(* CODESYS project xlh_transport_trolley_ST_00_90.project
   Description: Receives some incoming messages and echoes them with CAN-ID +1
   Company: 3S - Smart Software Solutions GmbH
   Version: 1.0.0.0
   Title: CAN Bus API Example
   Author: 3S - Smart Software Solutions GmbH

Project tree, tasks and I/O mapping:
  xlh_base : CODESYS Control for Raspberry Pi 64 SL, CODESYS, order no. 2302000009, version 4.18.0.0
    application app
      libraries: Standard, 3.5.18.0 (System); Util, 3.5.21.0 (System); VisuDialogs, * (System); Memory, * (3S - Smart Software Solutions GmbH); CmpBitmapPool, * (System)
      task MAIN_TASK (cyclic, interval 5 ms, priority 0) calls MAIN
      task VISU_TASK (cyclic, interval 100 ms, priority 31) calls VisuElems.Visu_Prg
      FSM/
        program TW_ST [ST]
        data type eTW
      visualisation VISU_SIMU
      function block FB_SIMU_TW [ST]
      image pool ImagePool
      program MAIN [ST]
      Depictor
      function block FB_XLH_GPIO [CFC]
    SoftMotion General Axis Pool
      a_axis : SM_Drive_PosControl, CODESYS, order no. 1805, version 4.18.0.0
          settings: wDriveID = 4; dwRatioTechUnitsDenom = 101846; iRatioTechUnitsNum = -125; eRampType = 1; fSWMaxVelocity = 50; fSWMaxAcceleration = 100; fSWMaxDeceleration = 100; fSWMaxJerk = 1000; fSWLimitNegative = -1000.0; ScalingIncs = 814768; ScalingUnits = 1000; InvertDirection = TRUE; IsLinearMotor = TRUE; MaximumOutputVelocityInt = 40738; MinimumOutputVelocityInt = -40738; Kp = 0.05; MaxFollowingError = 5.0; EnableFollowingErrorCheck = TRUE; DeadTime = 3.0
      x_axis : SM_Drive_PosControl, CODESYS, order no. 1805, version 4.18.0.0
          settings: dwRatioTechUnitsDenom = 101846; iRatioTechUnitsNum = 125; eRampType = 1; fSWMaxVelocity = 50; fSWMaxAcceleration = 100; fSWMaxDeceleration = 100; fSWMaxJerk = 1000; fSWLimitNegative = -1000; ScalingIncs = 814768; ScalingUnits = 1000; IsLinearMotor = TRUE; MaximumOutputVelocityInt = 40738; MinimumOutputVelocityInt = -40738; Kp = 0.05; MaxFollowingError = 5.0; EnableFollowingErrorCheck = TRUE; DeadTime = 3.0
      y_axis : SM_Drive_PosControl, CODESYS, order no. 1805, version 4.18.0.0
          settings: wDriveID = 2; dwRatioTechUnitsDenom = 101846; iRatioTechUnitsNum = 125; eRampType = 1; fSWMaxVelocity = 50; fSWMaxAcceleration = 100; fSWMaxDeceleration = 100; fSWMaxJerk = 1000; fSWLimitNegative = -1000; ScalingIncs = 814768; ScalingUnits = 1000; IsLinearMotor = TRUE; MaximumOutputVelocityInt = 40738; MinimumOutputVelocityInt = -40738; Kp = 0.05; MaxFollowingError = 5.0; EnableFollowingErrorCheck = TRUE; DeadTime = 3.0
      z_axis : SM_Drive_PosControl, CODESYS, order no. 1805, version 4.18.0.0
          settings: wDriveID = 3; dwRatioTechUnitsDenom = 101846; iRatioTechUnitsNum = 125; eRampType = 1; fSWMaxVelocity = 50; fSWMaxAcceleration = 100; fSWMaxDeceleration = 100; fSWMaxJerk = 1000; fSWLimitNegative = -1000; ScalingIncs = 814768; ScalingUnits = 1000; IsLinearMotor = TRUE; MaximumOutputVelocityInt = 40738; MinimumOutputVelocityInt = -40738; Kp = 0.05; MaxFollowingError = 5.0; EnableFollowingErrorCheck = TRUE; DeadTime = 3.0
    GPIOs_A_B : GPIOs B+/Pi2, CODESYS, version 4.18.0.0
        input  app.MAIN.gpio.bSw1 : BOOL  // digital inputs (GPIO0..GPIO31).Bit4
        input  app.MAIN.gpio.bSw2 : BOOL  // digital inputs (GPIO0..GPIO31).Bit5
        input  app.MAIN.gpio.bSw3 : BOOL  // digital inputs (GPIO0..GPIO31).Bit6
        input  app.MAIN.gpio.bSw4 : BOOL  // digital inputs (GPIO0..GPIO31).Bit12
        input  app.MAIN.gpio.bSw5 : BOOL  // digital inputs (GPIO0..GPIO31).Bit13
        input  app.MAIN.gpio.bSw6 : BOOL  // digital inputs (GPIO0..GPIO31).Bit16
        input  app.MAIN.gpio.bSw7 : BOOL  // digital inputs (GPIO0..GPIO31).Bit17
        input  app.MAIN.gpio.bSw8 : BOOL  // digital inputs (GPIO0..GPIO31).Bit19
        output app.MAIN.gpio.bLed1 : BOOL  // digital outputs (GPIO0..GPIO31).Bit20
        output app.MAIN.gpio.bLed2 : BOOL  // digital outputs (GPIO0..GPIO31).Bit21
        output app.MAIN.gpio.bLed3 : BOOL  // digital outputs (GPIO0..GPIO31).Bit22
        output app.MAIN.gpio.bLed4 : BOOL  // digital outputs (GPIO0..GPIO31).Bit23
        output app.MAIN.gpio.bLed5 : BOOL  // digital outputs (GPIO0..GPIO31).Bit24
        output app.MAIN.gpio.bLed6 : BOOL  // digital outputs (GPIO0..GPIO31).Bit26
        output app.MAIN.gpio.bLed7 : BOOL  // digital outputs (GPIO0..GPIO31).Bit27
        unmapped channels: digital inputs (GPIO0..GPIO31), digital outputs (GPIO0..GPIO31)
    Onewire
    Camera device
      <Leer>
    SPI
    I²C
  libraries: VisuSymbols, 4.5.0.0 (System); DepictorBase, 1.2.0.0 (CODESYS); DepictorBase, * (CODESYS)
  text list GlobalTextList
  5ce3da45-db07-42e7-a21c-a00fff4ed8f6|Transportwagen.drawio.png
*)

// xlh_base/app/FSM/eTW
{attribute 'qualified_only'}
{attribute 'strict'}
TYPE eTW :
(
	STARTUP := 0,
	WARTE_START := 10,
	WAGEN_RICHTUNG_BELADEN := 20,
	WAGEN_BELADEN := 30,
	WAGEN_ENTLADEN := 40,
	WAGEN_RICHTUNG_ENTLADEN := 50,
	STOERUNG := 60
);
END_TYPE

// xlh_base/app/MAIN
PROGRAM MAIN 
VAR_INPUT
	
END_VAR
VAR	
	gpio: FB_XLH_GPIO;	
	fbSimuTw: FB_SIMU_TW;
END_VAR

// Zuweisung der Eingänge
TW_ST.bSF1_Start := gpio.bSw5;
TW_ST.bSF2_Stopp := NOT gpio.bSw6;
TW_ST.bFC1_Motorschutzschalter := gpio.bSw1;

// Aufruf Simulator Transportwagen
fbSimuTw.bMB1_VentilSilo := TW_ST.bMB1_VentilSilo;
fbSimuTw.bMB2_VentilLeeren := TW_ST.bMB2_VentilLeeren;
fbSimuTw.bKF1_MotorNachEntladen := TW_ST.bKF1_MotorNachEntladen;
fbSimuTw.bKF2_MotorNachBeladen := TW_ST.bKF2_MotorNachBeladen;
fbSimuTw();
TW_ST.bSF3_StellungEntladen := fbSimuTw.bSF3_StellungEntladen;
TW_ST.bSF4_StellungBeladen := fbSimuTw.bSF4_StellungBeladen;
// Aufruf der Prozesslogik
TW_ST();

// Zuweisung der Ausgänge
gpio.bLed1 := TW_ST.bEA1_LampeStoerung;
gpio.bLed2 := TW_ST.bMB1_VentilSilo;
gpio.bLed3 := TW_ST.bMB2_VentilLeeren;
gpio.bLed4 := TW_ST.bKF1_MotorNachEntladen;
gpio.bLed5 := TW_ST.bKF2_MotorNachBeladen;

END_PROGRAM

// xlh_base/app/FSM/TW_ST
PROGRAM TW_ST
VAR_INPUT
	bSF1_Start: BOOL;
	bSF2_Stopp: BOOL;
	bSF3_StellungEntladen: BOOL;
	bSF4_StellungBeladen: BOOL;
	bFC1_Motorschutzschalter: BOOL;
END_VAR
VAR_OUTPUT
	bEA1_LampeStoerung: BOOL;
	bMB1_VentilSilo: BOOL;
	bMB2_VentilLeeren: BOOL;
	bKF1_MotorNachEntladen: BOOL;
	bKF2_MotorNachBeladen: BOOL;
END_VAR
VAR
	eStatus: eTW;
	fbRtSF1_Start: R_TRIG;
	fbTonBeladen: TON;
	fbTonEntladen: TON;
END_VAR

// Erfassung der Signalflanken
fbRtSF1_Start(CLK:=bSF1_Start);
// Zeitelemente
fbTonBeladen(IN:=(eStatus = eTW.WAGEN_BELADEN), PT:=T#3S);
fbTonEntladen(IN:=(eStatus = eTW.WAGEN_ENTLADEN), PT:=T#2.5S);

// stoppen der Bewegung
IF NOT bSF2_Stopp AND eStatus <> eTW.STOERUNG THEN
	eStatus := eTW.WARTE_START;
END_IF

// Motorschutz
IF NOT bFC1_Motorschutzschalter THEN
	eStatus := eTW.STOERUNG;
END_IF

// Zustandsautomat
CASE eStatus OF
	eTW.STARTUP:
		eStatus := eTW.WARTE_START;
	
	eTW.WARTE_START:
		IF fbRtSF1_Start.Q THEN
			IF NOT bSF3_StellungEntladen THEN
				eStatus := eTW.WAGEN_RICHTUNG_BELADEN;
			ELSE
				// Resetierung nach Unterbruch
				eStatus := eTW.WAGEN_RICHTUNG_ENTLADEN;
			END_IF
		END_IF
		
	eTW.WAGEN_RICHTUNG_BELADEN:
		IF NOT bSF4_StellungBeladen THEN
			eStatus := eTW.WAGEN_BELADEN;
		END_IF
		
	eTW.WAGEN_BELADEN:
		IF fbTonBeladen.Q THEN
			eStatus := eTW.WAGEN_RICHTUNG_ENTLADEN;
		END_IF
		
	eTW.WAGEN_RICHTUNG_ENTLADEN:
		IF NOT bSF3_StellungEntladen THEN
			eStatus := eTW.WAGEN_ENTLADEN;
		END_IF
		
	eTW.WAGEN_ENTLADEN:
		IF fbTonEntladen.Q THEN
			eStatus := eTW.WARTE_START;
		END_IF
	
	eTW.STOERUNG:
		IF bSF2_Stopp AND bFC1_Motorschutzschalter THEN
			eStatus := eTW.WARTE_START;
		END_IF
		
	ELSE
		; // Fehler im Zustandsautomaten
END_CASE

bEA1_LampeStoerung := (eStatus = eTW.STOERUNG);
bMB1_VentilSilo := (eStatus = eTW.WAGEN_BELADEN);
bMB2_VentilLeeren := (eStatus = eTW.WAGEN_ENTLADEN);
bKF1_MotorNachEntladen := (eStatus = eTW.WAGEN_RICHTUNG_ENTLADEN);
bKF2_MotorNachBeladen := (eStatus = eTW.WAGEN_RICHTUNG_BELADEN);

END_PROGRAM

// xlh_base/app/FB_XLH_GPIO
FUNCTION_BLOCK FB_XLH_GPIO
VAR_INPUT
	bLed1: BOOL;
	bLed2: BOOL;
	bLed3: BOOL;
	bLed4: BOOL;
	bLed5: BOOL;
	bLed6: BOOL;
	bLed7: BOOL;	
END_VAR
VAR_OUTPUT
	bSw1: BOOL;
	bSw2: BOOL;
	bSw3: BOOL;
	bSw4: BOOL;
	bSw5: BOOL;
	bSw6: BOOL;
	bSw7: BOOL;
	bSw8: BOOL;
END_VAR

END_FUNCTION_BLOCK

// xlh_base/app/FB_SIMU_TW
FUNCTION_BLOCK FB_SIMU_TW
VAR_INPUT
	bMB1_VentilSilo: BOOL;
	bMB2_VentilLeeren: BOOL;
	bKF1_MotorNachEntladen: BOOL;
	bKF2_MotorNachBeladen: BOOL;
END_VAR
VAR_OUTPUT
	bSF3_StellungEntladen: BOOL;
	bSF4_StellungBeladen: BOOL;
	//
	rPosOffsetVentilSilo: REAL;
	rPosOffsetVentilTransportwagen: REAL;
	rPosOffsetTransportwagen: REAL;
	{attribute 'displaymode':='hex'}
	udiColorEsBeladen: UDINT;
	{attribute 'displaymode':='hex'}
	udiColorEsEntladen: UDINT;
	bTransportwagenInhaltVisible: BOOL;
END_VAR
VAR
	bStartup: BOOL := TRUE;
	fbTonTwInhaltShow: TON;
	fbTonTwInhaltHide: TON;
END_VAR

IF bStartup THEN
	bStartup := FALSE;
	rPosOffsetTransportwagen := -150.0;
END_IF

IF bMB1_VentilSilo THEN
	rPosOffsetVentilSilo := 25.0;
ELSE
	rPosOffsetVentilSilo := 0.0;
END_IF

IF bMB2_VentilLeeren THEN
	rPosOffsetVentilTransportwagen := 20.0;
ELSE
	rPosOffsetVentilTransportwagen := 0.0;
END_IF

IF bKF1_MotorNachEntladen THEN
	rPosOffsetTransportwagen := rPosOffsetTransportwagen - 1;
END_IF
IF bKF2_MotorNachBeladen THEN
	rPosOffsetTransportwagen := rPosOffsetTransportwagen + 1;
END_IF
rPosOffsetTransportwagen := LIMIT(-150.0, rPosOffsetTransportwagen, 150.0);

IF rPosOffsetTransportwagen >= 150.0 THEN
	bSF4_StellungBeladen := FALSE;
	udiColorEsBeladen := 16#FF00FF00;
ELSE
	bSF4_StellungBeladen := TRUE;
	udiColorEsBeladen := 16#FFA0A0A0;
END_IF

IF rPosOffsetTransportwagen <= -150.0 THEN
	bSF3_StellungEntladen := FALSE;
	udiColorEsEntladen := 16#FF00FF00;
ELSE
	bSF3_StellungEntladen := TRUE;
	udiColorEsEntladen := 16#FFA0A0A0;
END_IF

fbTonTwInhaltShow(IN:=NOT bSF4_StellungBeladen AND bMB1_VentilSilo,
	              PT:=T#2.9S);
IF fbTonTwInhaltShow.Q THEN
	bTransportwagenInhaltVisible := TRUE;
END_IF

fbTonTwInhaltHide(IN:=NOT bSF3_StellungEntladen,
	              PT:=T#2.4S);
IF fbTonTwInhaltHide.Q THEN
	bTransportwagenInhaltVisible := FALSE;
END_IF

END_FUNCTION_BLOCK

// xlh_base/app/VISU_SIMU
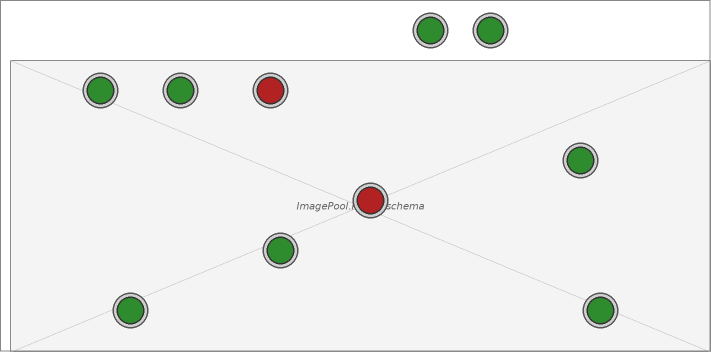
VISUALIZATION VISU_SIMU  // 711x352
    Image (10,60 701x292), image: ImagePool.Prinzipschema
    Lamp1 (80,70 41x41), variable: TW_ST.bSF1_Start, style: Lamp-Lamp1-Green
    Lamp1 (160,70 41x41), variable: TW_ST.bSF2_Stopp, style: Lamp-Lamp1-Green
    Lamp1 (250,70 41x41), variable: NOT TW_ST.bFC1_Motorschutzschalter, style: Lamp-Lamp1-Red
    Lamp1 (410,10 41x41), variable: TW_ST.bKF1_MotorNachEntladen, style: Lamp-Lamp1-Green
    Lamp1 (470,10 41x41), variable: TW_ST.bKF2_MotorNachBeladen, style: Lamp-Lamp1-Green
    Lamp1 (560,140 41x41), variable: TW_ST.bMB1_VentilSilo, style: Lamp-Lamp1-Green
    Lamp1 (110,290 41x41), variable: TW_ST.bSF3_StellungEntladen, style: Lamp-Lamp1-Green
    Lamp1 (580,290 41x41), variable: TW_ST.bSF4_StellungBeladen, style: Lamp-Lamp1-Green
    Lamp1 (350,180 41x41), variable: TW_ST.bEA1_LampeStoerung, style: Lamp-Lamp1-Red
    Lamp1 (260,230 41x41), variable: TW_ST.bMB2_VentilLeeren, style: Lamp-Lamp1-Green
END_VISUALIZATION
